SUBAPPLICATION QX_sim (* Subapplication Type *)
  (* Standard: 61499-2 *)
  (* Version 1.0, 2019-11-08, dorofeev *)
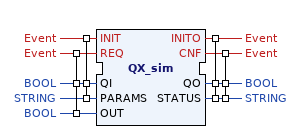
  EVENT_INPUT
    INIT WITH QI, PARAMS; (* Initialization Request *)
    REQ WITH QI, OUT; (* Normal Execution Request *)
  END_EVENT
  EVENT_OUTPUT
    INITO WITH QO, STATUS; (* Initialization Confirm *)
    CNF WITH QO, STATUS; (* Execution Confirmation *)
  END_EVENT
  VAR_INPUT
    QI : BOOL; (* Input event qualifier *)
    PARAMS : STRING;
    OUT : BOOL;
  END_VAR
  VAR_OUTPUT
    QO : BOOL; (* Output event qualifier *)
    STATUS : STRING;
  END_VAR
  EVENT_CONNECTIONS
    INIT TO INITO;
    REQ TO CNF;
  END_CONNECTIONS
  DATA_CONNECTIONS
    OUT TO QO;
  END_CONNECTIONS
END_SUBAPPLICATION
